{attribute 'Tc2GvlVarNames'}
VAR_GLOBAL
	Array_LPB_TDA_INT AT%MB1000: ARRAY[0..20] OF INT;
	Array_INT_Test : ARRAY [0..20] OF INT;
END_VAR

(* stored: Version 1.1.0.1, ProductVersion 3.1.4024.12
   GVL GVL_ADS: Id {7c90d152-c468-41b1-bae6-45b878c4775b} *)
